(* PLC project Unnamed, Unknown Unnamed 1 *)
(* stored: creationDateTime 2026-04-04T10:00:38, modificationDateTime 2026-04-04T10:00:38 *)

PROGRAM main
  VAR
    CRAC_Fan_Status : BOOL;
    Temp_High_Alarm : BOOL;
  END_VAR

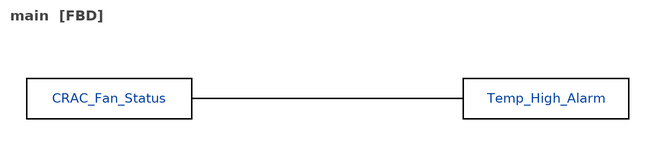
(* FBD diagram, written out as Structured Text *)
Temp_High_Alarm := CRAC_Fan_Status;
END_PROGRAM

CONFIGURATION Config0
  RESOURCE Res0 ON PLC
    TASK task0(INTERVAL := T#20ms, PRIORITY := 1);
    PROGRAM instance0 WITH task0 : main;
  END_RESOURCE
END_CONFIGURATION
